PROGRAM PRG_TcUnitMain
VAR
// Enable the test FBs to RUN TcUnit
	//fbTest_AteqControl	: FB_Test_AteqControl;
	//fbTest_ValveBank 		: FB_Test_ValveBank;

END_VAR


	//TcUnit.RUN_IN_SEQUENCE();

END_PROGRAM

(* stored: Version 1.1.0.1
   POU PRG_TcUnitMain: Id {17166b4e-59dc-4826-b23b-b13d729fc1f3}, SpecialFunc None *)
